// Mitsubishi GX Works2 project: 延时开关定时器   PLC: FX3U/FX3UC

PROGRAM MAIN
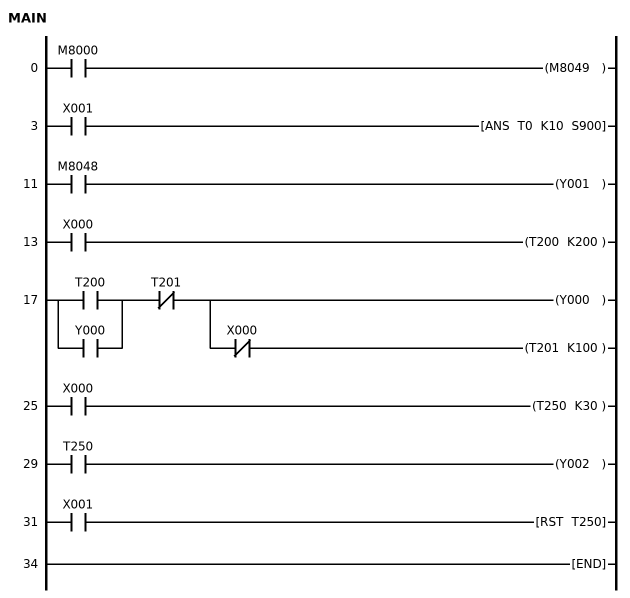
0     LD      M8000
      OUT     M8049
3     LD      X001
      ANS     T0 K10 S900
11    LD      M8048
      OUT     Y001
13    LD      X000
      OUT     T200 K200
17    LD      T200
      OR      Y000
      ANI     T201
      OUT     Y000
      ANI     X000
      OUT     T201 K100
25    LD      X000
      OUT     T250 K30
29    LD      T250
      OUT     Y002
31    LD      X001
      RST     T250
34    END
END_PROGRAM
